{attribute 'qualified_only'}
VAR_GLOBAL
	bInAckSignal		AT %I* 	: BOOL := TRUE;
	bEStop				AT %I*	: BOOL := FALSE;
END_VAR

(* stored: Version 1.1.0.1, ProductVersion 3.1.4024.12
   GVL GVL_Safety_IO: Id {055e14b0-3761-4718-92b0-a08f1db8711d} *)
